Fanuc KAREL source: ko00052.KL

-- PROVISIONAL review KL for V1013-1; original PC SHA256 1fe017fca780d53e8b25d9371e88d9abc334fc374a9ae1bd888ccda6f298e10f
-- Incomplete behavior may be omitted. Consult companion uncertainty JSON. Do not deploy.
PROGRAM KO00052
%NOLOCKGROUP
BEGIN
  -- UNRESOLVED_PC offsets 5-12; opcodes 9D,23
  -- UNRESOLVED_PC offsets 17-66; opcodes 27,27,49,7E,AD,22,1C,22,31,7E,4A
  -- UNRESOLVED_PC offsets 71-75; opcodes 7F
END KO00052
